# EPICS autosave request: ATTOCUBE/iocBoot/iocATTOCUBE-IOC-01/ATTOCUBE_01_axis_settings.req
# Attocube specific settings for an axis
$(P)$(IOCNAME):ACT$(AXIS):CMD:WR_AMPL.VAL
